PROGRAM MAIN
VAR
	al : Alarm;
	a2 : Alarm;
	
	raise: BOOL;
	confirm : BOOL;
	clear : BOOL;
	
	raise2: BOOL;
	confirm2 : BOOL;
	clear2 : BOOL;
	
	clearAlarms : BOOL; 
	fbEventLogger : FB_TcEventLogger;
	iEventLoggerSetting : I_TcClearLoggedEventsSettings;
	fbEventLoggerSetting : FB_TcClearLoggedEventsSettings;
END_VAR

al(
	AlarmID := TC_Events.Alarm.Event,
	bRaiseAlarm := raise);

a2(
	AlarmID := TC_Events.Alarm.AlarmEvent2,
	bRaiseAlarm := raise2);
clearAlarms := HMI.clearAlarmAll;	
FB_ExportCSV(bExport := HMI.bExportCSV);
ClearLoggedEvent(HMI.clearlogged);

METHOD ClearLoggedEvent : BOOL
VAR_INPUT
	bClearLoggedEvent : BOOL;
END_VAR

VAR
	
	clear : BOOL;
END_VAR
IF bClearLoggedEvent THEN
	fbEventLoggerSetting.Clear();
	//fbEventLogger.ClearAllAlarms(0, bClearLoggedEvent);	
	fbEventLogger.ConfirmAllAlarms(0);
	clearAlarms := TRUE;
	FB_ExportCSV(bExport := TRUE);	
	fbEventLogger.ClearLoggedEvents(fbEventLoggerSetting);
	bClearLoggedEvent := FALSE;
	
END_IF
END_METHOD

END_PROGRAM

(* stored: Version 1.1.0.1, ProductVersion 3.1.4024.6
   POU MAIN: Id {e24e4ddb-35a4-44b0-8037-fc097a3e01d2}, SpecialFunc None
   Method ClearLoggedEvent: Id {2fe84791-1de5-46cc-acc5-006b30e4015a} *)
